// LS Electric XG5000 project: 김동혁
// PLC NewPLC
// module base 0 slot 0: 입출력 모듈:XBC-DR32H (DC 24V 입력, 릴레이 출력 32점)

PROGRAM NewProgram (task: 스캔 프로그램)

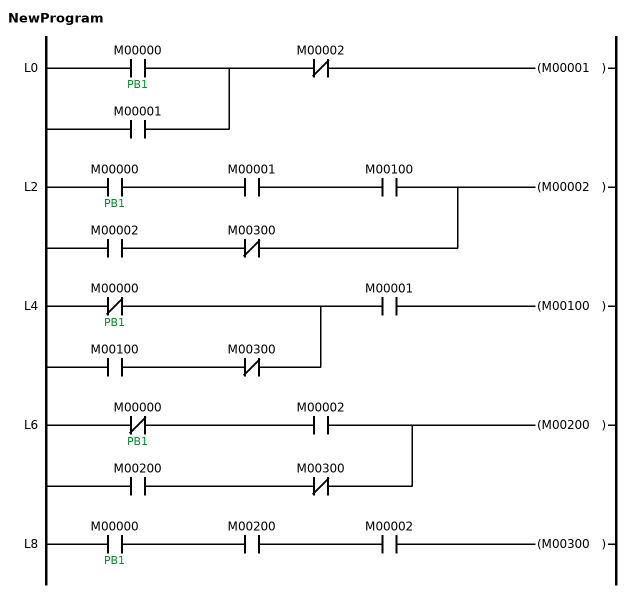
; L0
LOAD      M00000	// PB1
OR        M00001
AND NOT   M00002
OUT       M00001
; L2
LOAD      M00000	// PB1
AND       M00001
AND       M00100
LOAD      M00002
AND NOT   M00300
OR LOAD
OUT       M00002
; L4
LOAD NOT  M00000	// PB1
LOAD      M00100
AND NOT   M00300
OR LOAD
AND       M00001
OUT       M00100
; L6
LOAD NOT  M00000	// PB1
AND       M00002
LOAD      M00200
AND NOT   M00300
OR LOAD
OUT       M00200
; L8
LOAD      M00000	// PB1
AND       M00200
AND       M00002
OUT       M00300

VARIABLES AND COMMENTS (devices not used above)
M10000	BIT	rl